TYPE ST_ValveOutput_1 :
STRUCT
	bEnable					AT %Q* : BOOL := 0;
	nValveOutput 			AT %Q* : INT := 19660;
END_STRUCT
END_TYPE

(* stored: Version 1.1.0.1, ProductVersion 3.1.4024.12
   DUT ST_ValveOutput_1: Id {d3799cdb-f9fc-4361-8785-23f42470728a} *)
